INTERFACE IOutputDevice EXTENDS IDevice

METHOD UpdateOutputsFromState
END_METHOD

END_INTERFACE

(* stored: Version 1.1.0.1
   Itf IOutputDevice: Id {ac0084c1-bfc2-4478-a358-5412fb85e829}
   Method UpdateOutputsFromState: Id {c47b5cfd-628e-4cc0-a4d5-0e13fe24adee} *)
